FUNCTION_BLOCK ExerciseCirculationPumpsParametersFB
VAR_INPUT
END_VAR
VAR_OUTPUT
END_VAR
VAR
END_VAR

END_FUNCTION_BLOCK

(* stored: Version 1.1.0.1, ProductVersion 3.1.4024.6
   POU ExerciseCirculationPumpsParametersFB: Id {221f950b-bc06-4040-9983-aa363eb5fa79}, SpecialFunc None *)
